{attribute 'qualified_only'}
{attribute 'strict'}
TYPE EFeedbackMsgPlc :
(
	SmokeDetectedMsg := 0,
	SmokeDetectorFaultMsg,
	VacuumDetectorMsg,
	AmsNetIdMsg
);
END_TYPE

(* stored: Version 1.1.0.1, ProductVersion 3.1.4024.12
   DUT EFeedbackMsgPlc: Id {3d86c321-fa97-473c-8691-d6cf9426eef1} *)
